{attribute 'no_explicit_call' := 'FB_EventSubscriber is a CLASS and must be accessed using methods or properties'}
FUNCTION_BLOCK FB_EventSubscriber IMPLEMENTS I_Observer
VAR	
	_eventPublisher					: I_EventPublisher;
	_event							: INT;
	
	verbose							: BOOL := TRUE;

	// Register after online change 
	registeredAtPublisher			: BOOL;	
END_VAR


// The body of a class must not be used for code.  
// Cyclic code should be called from a method if needed.

METHOD ChangePublisher
VAR_INPUT
	eventPublisher					: I_EventPublisher;
END_VAR
_eventPublisher := eventPublisher;
END_METHOD

METHOD cyclicCall
// Did we already register in the publisher?
IF NOT registeredAtPublisher	THEN
	registeredAtPublisher := _eventPublisher.attach(THIS^);
END_IF
END_METHOD

// IMPLEMENTED ONLY FOR TESTING PURPOSES
PROPERTY Event : int
GET
event := _event;
END_GET
END_PROPERTY

METHOD FB_init : BOOL
VAR_INPUT
	bInitRetains	 				: BOOL; // if TRUE, the retain variables are initialized (warm start / cold start)
	bInCopyCode 					: BOOL;  // if TRUE, the instance afterwards gets moved into the copy code (online change)
	EventPublisher					: I_EventPublisher;
END_VAR
_eventPublisher := eventPublisher;
END_METHOD

METHOD PRIVATE message : BOOL
VAR_INPUT
	dintArg						: DINT;
END_VAR
// Log message
IF verbose  THEN
	ADSLOGDINT(
		msgCtrlMask := ADSLOG_MSGTYPE_HINT OR ADSLOG_MSGTYPE_LOG, // ADSLOG_MSGTYPE_ERROR OR ADSLOG_MSGTYPE_LOG, 
		msgFmtStr 	:= 'Subscriber 1 knows the value changed to %d',
		dintArg 	:= dintArg
		);
END_IF
END_METHOD

METHOD Update : BOOL
// the publisher mentions an update, fetch the data
_event := _eventPublisher.event;
message(TO_DINT(_event));
END_METHOD

END_FUNCTION_BLOCK

(* stored: Version 1.1.0.1, ProductVersion 3.1.4024.12
   POU FB_EventSubscriber: Id {d4dce0f2-3ded-43b2-8491-9014ab19c774}, SpecialFunc None
   Method ChangePublisher: Id {5d3a73b4-e70f-47cf-85f0-6c2314916a13}
   Method cyclicCall: Id {5c9ecd9a-07d4-463a-ade9-6bde0f93e10b}
   Property Event: Id {aa9553a2-33bf-40d8-a234-28f7162b10c5}
   Get Get: Id {231fdd1c-03f2-4591-b73d-451501ccc307}
   Method FB_init: Id {3bae645b-cda2-435b-a713-7a36da169a78}
   Method message: Id {e4f26ffc-57fb-4c96-b5ee-4b9c9356b25c}
   Method Update: Id {26657e55-00fd-4c13-80e1-21813364b2ff} *)
